(* CODESYS project PLCTEST.project
   Title: PLCTEST
   Author: Peter
   Version: 0.0.0.13

Project tree, tasks and I/O mapping:
  MyController_1 : TM241CEC24T/U, Schneider Electric, order no. TM241CEC24T/U, version 4.0.6.18
    application Application
      libraries: HMISCU PTOPWM, 2.0.1.4 (Schneider Electric); SM3_Basic, 3.5.3.83 (3S - Smart Software Solutions GmbH); CANmotion Lexium Library, 1.3.1.0 (Schneider Electric)
      task MAST (cyclic, interval 2 ms, priority 15, watchdog 100 ms x 1) calls POU_TEST
      program POU_TEST [ST]
      global variables GVL
      program POU [CFC]
    DI : Digital Inputs, Schneider Electric, version 4.0.6.18
        input  iwDI_IW0 : WORD  // IW0
        input  ibDI_IB1 : BYTE  // IB1
    DQ : Digital Outputs, Schneider Electric, version 4.0.6.18
        output Application.POU_TEST.q0 : BOOL  // QW0.Q0
        output Application.POU_TEST.q1 : BOOL  // QW0.Q1
        output Application.POU_TEST.q2 : BOOL  // QW0.Q2
        output Application.POU_TEST.q0 : BOOL  // QW0.Q4
        output Application.POU_TEST.q1 : BOOL  // QW0.Q5
        output Application.POU_TEST.q2 : BOOL  // QW0.Q6
        output Application.POU_TEST.q0 : BOOL  // QW0.Q8
        output Application.POU_TEST.q1 : BOOL  // QW0.Q9
        unmapped channels: QW0, QB1
    Counters : Counters, Schneider Electric, version 4.0.6.18
    Pulse_Generators : Pulse Generators, Schneider Electric, version 4.0.6.18
    Cartridge_1 : Cartridge, Schneider Electric, version 4.0.6.18
    IO_Bus : IO bus - TM3, Schneider Electric, version 4.0.6.18
      Module_1 : TM3SAF5R/G, Schneider Electric, order no. TM3SAF5R/G, version 1.0.1.12
          input  iwModule_1_IW0 : WORD  // IW0
          output qbModule_1_QB0 : BYTE  // QB0
      Module_2 : TM3AQ4/G, Schneider Electric, order no. TM3AQ4/G, version 1.0.0.12
          output qiModule_2_QW0 : INT  // QW0
          output qiModule_2_QW1 : INT  // QW1
          output qiModule_2_QW2 : INT  // QW2
          output qiModule_2_QW3 : INT  // QW3
          input  ibModule_2_IBStatusQW0 : BYTE  // IBStatusQW0
          input  ibModule_2_IBStatusQW1 : BYTE  // IBStatusQW1
          input  ibModule_2_IBStatusQW2 : BYTE  // IBStatusQW2
          input  ibModule_2_IBStatusQW3 : BYTE  // IBStatusQW3
    COM_Bus : COM bus, Schneider Electric, version 4.0.6.18
    Ethernet_1 : Ethernet Network, Schneider Electric, version 4.0.6.18
    Serial_Line_1 : Serial line, Schneider Electric, version 4.0.6.18
      SoMachine_Network_Manager1 : SoMachine-Network Manager, Schneider Electric, version 4.0.0.2
    Serial_Line_2 : Serial line, Schneider Electric, version 4.0.6.18
      Modbus_Manager1 : Modbus Manager, Schneider Electric, version 4.0.0.2
    CAN_1 : CANopen bus, Schneider Electric, version 4.0.6.18
      CANopen_Performance : CANopen Performance, Schneider Electric, order no. 1806, version 3.0.1.24
          settings: Heartbeat in Milliseconds = 100; ConfigVersion = 50659584
        Lexium_32_M : Lexium 32 M, Schneider Electric, order no. 91200, version 3.5.9.0
            settings: General Options.Optional Device = TRUE; NODEIDSAVED = 1; SDO Timeout = 1000000; Explicit Deactivate PDOs = FALSE; EXPERTSETTINGS = False; Nodeguarding.Guard Time = 100 ms; Heartbeat-Producer Time = 200; PDO 16#1400.COBID = 16#0201; PDO 16#1801.COBID = 16#C0000281; Generic COBID = '$NODEID+16#C0000280'; PDO 16#1802.COBID = 16#C0000381; Generic COBID = '$NODEID+16#C0000380'; PDO 16#1803.COBID = 16#C0000481; Generic COBID = '$NODEID+16#C0000480'; Heartbeat-Consuming1.Heartbeat-Time = 300 ms; Controlword.Subindex = 16#00; Target position.Subindex = 16#00; Controlword.Subindex = 16#00; Target velocity.Subindex = 16#00; Statusword.Subindex = 16#00; Position actual value.Subindex = 16#00; Statusword.Subindex = 16#00; Velocity actual value.Subindex = 16#00; SDO List.Set Guardtime.Index = 16#100C; SDO List.Set Guardtime.Subindex = 16#00; SDO List.Set Guardtime.Value = 16#00000064; SDO List.Set Guardtime.Size = 16; SDO List.Set Guardtime.AbortIfError = FALSE; SDO List.Set Guardtime.JumpToLine = FALSE; SDO List.Set Guardtime.Line = 0; SDO List.Set Lifetime.Index = 16#100D; SDO List.Set Lifetime.Subindex = 16#00; SDO List.Set Lifetime.Value = 16#00000000; SDO List.Set Lifetime.Size = 8; SDO List.Set Lifetime.AbortIfError = FALSE; SDO List.Set Lifetime.JumpToLine = FALSE; SDO List.Set Lifetime.Line = 0; SDO List.Disable Emcy CobID.Index = 16#1014; SDO List.Disable Emcy CobID.Subindex = 16#00; SDO List.Disable Emcy CobID.Value = 16#80000081;
              SDO List.Disable Emcy CobID.Size = 32; SDO List.Disable Emcy CobID.AbortIfError = FALSE; SDO List.Disable Emcy CobID.JumpToLine = FALSE; SDO List.Disable Emcy CobID.Line = 0; SDO List.Set Emcy CobID.Index = 16#1014; SDO List.Set Emcy CobID.Subindex = 16#00; SDO List.Set Emcy CobID.Value = 16#00000081; SDO List.Set Emcy CobID.Size = 32; SDO List.Set Emcy CobID.AbortIfError = FALSE; SDO List.Set Emcy CobID.JumpToLine = FALSE; SDO List.Set Emcy CobID.Line = 0; SDO List.Set Heartbeat Consumer.Index = 16#1016; SDO List.Set Heartbeat Consumer.Subindex = 16#01; SDO List.Set Heartbeat Consumer.Value = 16#007F012C; SDO List.Set Heartbeat Consumer.Size = 32; SDO List.Set Heartbeat Consumer.AbortIfError = FALSE; SDO List.Set Heartbeat Consumer.JumpToLine = FALSE; SDO List.Set Heartbeat Consumer.Line = 0; SDO List.Set Heartbeat Consumer.Index = 16#1016; SDO List.Set Heartbeat Consumer.Subindex = 16#02; SDO List.Set Heartbeat Consumer.Value = 0; SDO List.Set Heartbeat Consumer.Size = 32; SDO List.Set Heartbeat Consumer.AbortIfError = FALSE; SDO List.Set Heartbeat Consumer.JumpToLine = FALSE; SDO List.Set Heartbeat Consumer.Line = 0; SDO List.Set Heartbeat Consumer.Index = 16#1016; SDO List.Set Heartbeat Consumer.Subindex = 16#03; SDO List.Set Heartbeat Consumer.Value = 0; SDO List.Set Heartbeat Consumer.Size = 32; SDO List.Set Heartbeat Consumer.AbortIfError = FALSE; SDO List.Set Heartbeat Consumer.JumpToLine = FALSE; SDO List.Set Heartbeat Consumer.Line = 0; SDO List.Set Heartbeat Producer.Index = 16#1017; SDO List.Set Heartbeat Producer.Subindex = 16#00; SDO List.Set Heartbeat Producer.Value = 16#000000C8; SDO List.Set Heartbeat Producer.Size = 16; SDO List.Set Heartbeat Producer.AbortIfError = FALSE; SDO List.Set Heartbeat Producer.JumpToLine = FALSE; SDO List.Set Heartbeat Producer.Line = 0; SDO List.Disable PDO.Index = 16#1400;
              SDO List.Disable PDO.Subindex = 16#01; SDO List.Disable PDO.Value = 16#80000201; SDO List.Disable PDO.Size = 32; SDO List.Disable PDO.AbortIfError = FALSE; SDO List.Disable PDO.JumpToLine = FALSE; SDO List.Disable PDO.Line = 0; SDO List.Set transmission type.Index = 16#1400; SDO List.Set transmission type.Subindex = 16#02; SDO List.Set transmission type.Value = 16#FF; SDO List.Set transmission type.Size = 8; SDO List.Set transmission type.AbortIfError = FALSE; SDO List.Set transmission type.JumpToLine = FALSE; SDO List.Set transmission type.Line = 0; SDO List.Clear pdo mapping.Index = 16#1600; SDO List.Clear pdo mapping.Subindex = 16#00; SDO List.Clear pdo mapping.Value = 16#0; SDO List.Clear pdo mapping.Size = 8; SDO List.Clear pdo mapping.AbortIfError = FALSE; SDO List.Clear pdo mapping.JumpToLine = FALSE; SDO List.Clear pdo mapping.Line = 0; SDO List.Set Mapping.Index = 16#1600; SDO List.Set Mapping.Subindex = 16#01; SDO List.Set Mapping.Value = 16#301B1F10; SDO List.Set Mapping.Size = 32; SDO List.Set Mapping.AbortIfError = FALSE; SDO List.Set Mapping.JumpToLine = FALSE; SDO List.Set Mapping.Line = 0; SDO List.Set Mapping.Index = 16#1600; SDO List.Set Mapping.Subindex = 16#02; SDO List.Set Mapping.Value = 16#301B2210; SDO List.Set Mapping.Size = 32; SDO List.Set Mapping.AbortIfError = FALSE; SDO List.Set Mapping.JumpToLine = FALSE; SDO List.Set Mapping.Line = 0; SDO List.Set Mapping.Index = 16#1600; SDO List.Set Mapping.Subindex = 16#03; SDO List.Set Mapping.Value = 16#301B2120; SDO List.Set Mapping.Size = 32; SDO List.Set Mapping.AbortIfError = FALSE; SDO List.Set Mapping.JumpToLine = FALSE;
              SDO List.Set Mapping.Line = 0; SDO List.Set number of pdos.Index = 16#1600; SDO List.Set number of pdos.Subindex = 16#00; SDO List.Set number of pdos.Value = 16#03; SDO List.Set number of pdos.Size = 8; SDO List.Set number of pdos.AbortIfError = FALSE; SDO List.Set number of pdos.JumpToLine = FALSE; SDO List.Set number of pdos.Line = 0; SDO List.Set and enable COB-ID.Index = 16#1400; SDO List.Set and enable COB-ID.Subindex = 16#01; SDO List.Set and enable COB-ID.Value = 16#00000201; SDO List.Set and enable COB-ID.Size = 32; SDO List.Set and enable COB-ID.AbortIfError = FALSE; SDO List.Set and enable COB-ID.JumpToLine = FALSE; SDO List.Set and enable COB-ID.Line = 0; SDO List.Disable PDO.Index = 16#1401; SDO List.Disable PDO.Subindex = 16#01; SDO List.Disable PDO.Value = 16#80000301; SDO List.Disable PDO.Size = 32; SDO List.Disable PDO.AbortIfError = FALSE; SDO List.Disable PDO.JumpToLine = FALSE; SDO List.Disable PDO.Line = 0; SDO List.Disable PDO.Index = 16#1402; SDO List.Disable PDO.Subindex = 16#01; SDO List.Disable PDO.Value = 16#80000401; SDO List.Disable PDO.Size = 32; SDO List.Disable PDO.AbortIfError = FALSE; SDO List.Disable PDO.JumpToLine = FALSE; SDO List.Disable PDO.Line = 0; SDO List.Disable PDO.Index = 16#1403; SDO List.Disable PDO.Subindex = 16#01; SDO List.Disable PDO.Value = 16#80000501; SDO List.Disable PDO.Size = 32; SDO List.Disable PDO.AbortIfError = FALSE; SDO List.Disable PDO.JumpToLine = FALSE; SDO List.Disable PDO.Line = 0; SDO List.Disable PDO.Index = 16#1800; SDO List.Disable PDO.Subindex = 16#01; SDO List.Disable PDO.Value = 16#C0000181; SDO List.Disable PDO.Size = 32;
              SDO List.Disable PDO.AbortIfError = FALSE; SDO List.Disable PDO.JumpToLine = FALSE; SDO List.Disable PDO.Line = 0; SDO List.Set transmission type.Index = 16#1800; SDO List.Set transmission type.Subindex = 16#02; SDO List.Set transmission type.Value = 16#FF; SDO List.Set transmission type.Size = 8; SDO List.Set transmission type.AbortIfError = FALSE; SDO List.Set transmission type.JumpToLine = FALSE; SDO List.Set transmission type.Line = 0; SDO List.Set inhibit time.Index = 16#1800; SDO List.Set inhibit time.Subindex = 16#03; SDO List.Set inhibit time.Value = 16#0064; SDO List.Set inhibit time.Size = 16; SDO List.Set inhibit time.AbortIfError = FALSE; SDO List.Set inhibit time.JumpToLine = FALSE; SDO List.Set inhibit time.Line = 0; SDO List.Set event time.Index = 16#1800; SDO List.Set event time.Subindex = 16#05; SDO List.Set event time.Value = 16#0000; SDO List.Set event time.Size = 16; SDO List.Set event time.AbortIfError = FALSE; SDO List.Set event time.JumpToLine = FALSE; SDO List.Set event time.Line = 0; SDO List.Clear pdo mapping.Index = 16#1A00; SDO List.Clear pdo mapping.Subindex = 16#00; SDO List.Clear pdo mapping.Value = 16#0; SDO List.Clear pdo mapping.Size = 8; SDO List.Clear pdo mapping.AbortIfError = FALSE; SDO List.Clear pdo mapping.JumpToLine = FALSE; SDO List.Clear pdo mapping.Line = 0; SDO List.Set Mapping.Index = 16#1A00; SDO List.Set Mapping.Subindex = 16#01; SDO List.Set Mapping.Value = 16#301B2510; SDO List.Set Mapping.Size = 32; SDO List.Set Mapping.AbortIfError = FALSE; SDO List.Set Mapping.JumpToLine = FALSE; SDO List.Set Mapping.Line = 0; SDO List.Set Mapping.Index = 16#1A00; SDO List.Set Mapping.Subindex = 16#02;
              SDO List.Set Mapping.Value = 16#301B2610; SDO List.Set Mapping.Size = 32; SDO List.Set Mapping.AbortIfError = FALSE; SDO List.Set Mapping.JumpToLine = FALSE; SDO List.Set Mapping.Line = 0; SDO List.Set Mapping.Index = 16#1A00; SDO List.Set Mapping.Subindex = 16#03; SDO List.Set Mapping.Value = 16#301B2710; SDO List.Set Mapping.Size = 32; SDO List.Set Mapping.AbortIfError = FALSE; SDO List.Set Mapping.JumpToLine = FALSE; SDO List.Set Mapping.Line = 0; SDO List.Set Mapping.Index = 16#1A00; SDO List.Set Mapping.Subindex = 16#04; SDO List.Set Mapping.Value = 16#301B2810; SDO List.Set Mapping.Size = 32; SDO List.Set Mapping.AbortIfError = FALSE; SDO List.Set Mapping.JumpToLine = FALSE; SDO List.Set Mapping.Line = 0; SDO List.Set number of pdos.Index = 16#1A00; SDO List.Set number of pdos.Subindex = 16#00; SDO List.Set number of pdos.Value = 16#04; SDO List.Set number of pdos.Size = 8; SDO List.Set number of pdos.AbortIfError = FALSE; SDO List.Set number of pdos.JumpToLine = FALSE; SDO List.Set number of pdos.Line = 0; SDO List.Set and enable COB-ID.Index = 16#1800; SDO List.Set and enable COB-ID.Subindex = 16#01; SDO List.Set and enable COB-ID.Value = 16#40000181; SDO List.Set and enable COB-ID.Size = 32; SDO List.Set and enable COB-ID.AbortIfError = FALSE; SDO List.Set and enable COB-ID.JumpToLine = FALSE; SDO List.Set and enable COB-ID.Line = 0; SDO List.Disable PDO.Index = 16#1801; SDO List.Disable PDO.Subindex = 16#01; SDO List.Disable PDO.Value = 16#C0000281; SDO List.Disable PDO.Size = 32; SDO List.Disable PDO.AbortIfError = FALSE; SDO List.Disable PDO.JumpToLine = FALSE; SDO List.Disable PDO.Line = 0;
              SDO List.Disable PDO.Index = 16#1802; SDO List.Disable PDO.Subindex = 16#01; SDO List.Disable PDO.Value = 16#C0000381; SDO List.Disable PDO.Size = 32; SDO List.Disable PDO.AbortIfError = FALSE; SDO List.Disable PDO.JumpToLine = FALSE; SDO List.Disable PDO.Line = 0; SDO List.Disable PDO.Index = 16#1803; SDO List.Disable PDO.Subindex = 16#01; SDO List.Disable PDO.Value = 16#C0000481; SDO List.Disable PDO.Size = 32; SDO List.Disable PDO.AbortIfError = FALSE; SDO List.Disable PDO.JumpToLine = FALSE; SDO List.Disable PDO.Line = 0; SDO List.Automap SDO1.Index = 16#3041; SDO List.Automap SDO1.Subindex = 16#0B; SDO List.Automap SDO1.Value = 15; SDO List.Automap SDO1.Size = 16; SDO List.Automap SDO1.AbortIfError = FALSE; SDO List.Automap SDO1.JumpToLine = FALSE; SDO List.Automap SDO1.Line = 0; SDO List.Automap SDO2.Index = 16#301B; SDO List.Automap SDO2.Subindex = 16#08; SDO List.Automap SDO2.Value = 1; SDO List.Automap SDO2.Size = 16; SDO List.Automap SDO2.AbortIfError = FALSE; SDO List.Automap SDO2.JumpToLine = FALSE; SDO List.Automap SDO2.Line = 0; SDO List.Automap SDO2.Index = 16#301B; SDO List.Automap SDO2.Subindex = 16#1E; SDO List.Automap SDO2.Value = 10; SDO List.Automap SDO2.Size = 16; SDO List.Automap SDO2.AbortIfError = FALSE; SDO List.Automap SDO2.JumpToLine = FALSE; SDO List.Automap SDO2.Line = 0; ConfigVersion = 50659584
            unmapped channels: driveModeCtrl, RefA16, RefB32, driveStat, mfStat, motionStat, driveInput
*)

// MyController_1/Application/GVL
VAR_GLOBAL
END_VAR

// MyController_1/Application/POU_TEST
PROGRAM POU_TEST
VAR
	power_: INT;
	counter : INT := 0;
	lights : ARRAY [0..3] OF BOOL;
	q0 : BOOL;
	q1 : BOOL;
	q2 : BOOL;
	execute : BOOL;
	
	limit_1 : SEM_LXM.SetLimitSwitch_LXM;
	limit_2 : SEM_LXM.SetLimitSwitch_LXM;
	
	
	wordName : WORD;

	powerLXM : MC_Power_LXM;
	//power : SM3_Basic.MC_Power;
	motorJog : MC_Jog_LXM;
	mcReadParameter : MC_ReadAxisError_LXM;
	resetLXM : SEM_LXM.MC_Reset_LXM;
	power_1 : SEM_LXM.MC_Power_LXM;
	//stop : SM3_Basic.MC_Stop;
	//home : SM3_Basic.MC_Home;
	
	
	
	
	testOut :BOOL;


END_VAR

(*
//power.Enable := TRUE;
(*
powerLXM.Axis := Lexium_32_M;
motorJog.Axis := Lexium_32_M;*)
q0 := TRUE;
//resetLXM.

powerLXM.Enable := TRUE;
motorJog.Forward := TRUE;


//home.Execute:= TRUE;
powerLXM(Axis := Lexium_32_M);
//stop();
motorJog(Axis := Lexium_32_M);

*)
qbModule_1_QB0 := 0001;

mcReadParameter.Enable := TRUE;

wordName := mcReadParameter.ErrorID;
power_1.Enable := TRUE;

q1 := TRUE;

mcReadParameter(Axis := Lexium_32_M);

power_1(Axis := Lexium_32_M);
limit_1.LimitSwitch := 1;
limit_1.Mode := 0;

limit_1.Execute := execute;
limit_1(Axis := Lexium_32_M);

limit_2.LimitSwitch := 2;
limit_2.Mode := 0;
limit_2.Execute := execute;
limit_2(Axis := Lexium_32_M);

resetLXM(Axis := Lexium_32_M);



//motorJog.Forward := TRUE;
//motorJog.Fast := TRUE;
//motorJog.TipPos := 100;

motorJog(Axis := Lexium_32_M);

END_PROGRAM

// MyController_1/Application/POU
PROGRAM POU
VAR
	MC_Power_LXM_0: MC_Power_LXM;
	MC_ReadActualVelocity_LXM_0: MC_ReadActualVelocity_LXM;
	MC_MoveVelocity_LXM_0: MC_MoveVelocity_LXM;
	MC_Reset_LXM_0: MC_Reset_LXM;
	MC_ReadStatus_LXM_0 : MC_ReadStatus_LXM;
	xPower: BOOL;
	xReset: BOOL;
	MC_Stop_LXM_0: MC_Stop_LXM;
	xStop: BOOL;
	xMove: BOOL;
END_VAR

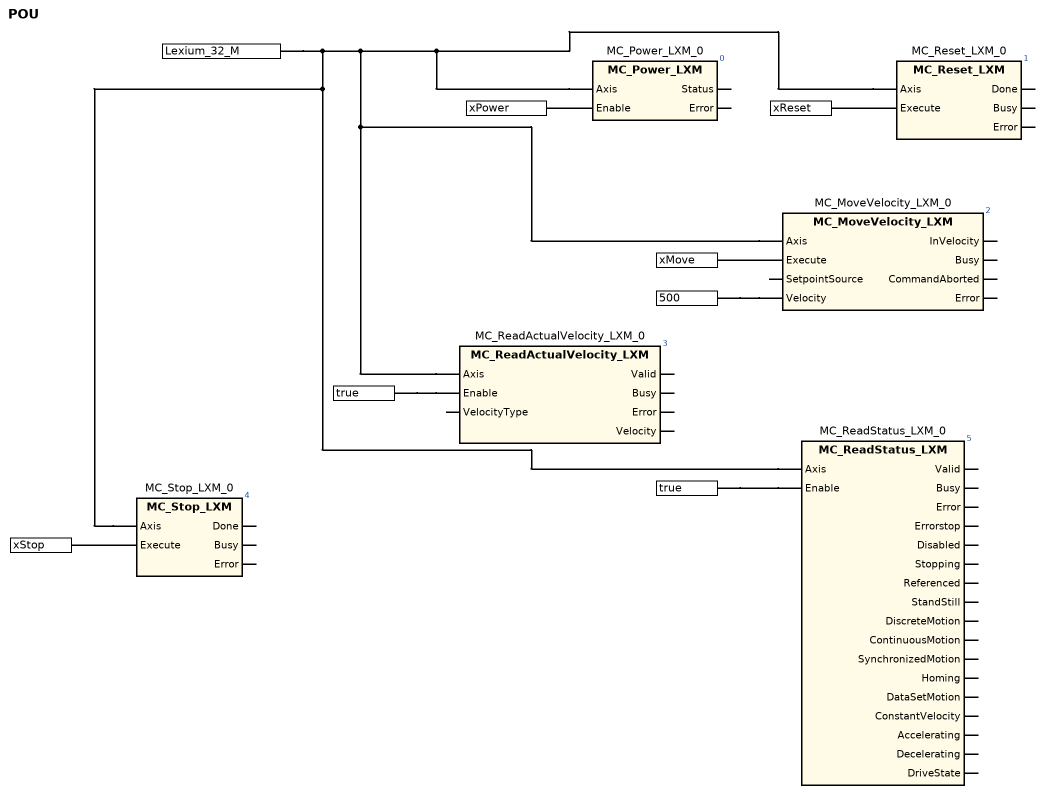
MC_Power_LXM_0(Axis := Lexium_32_M, Enable := xPower); // MC_Power_LXM
MC_Reset_LXM_0(Axis := Lexium_32_M, Execute := xReset); // MC_Reset_LXM
MC_MoveVelocity_LXM_0(Axis := Lexium_32_M, Execute := xMove, Velocity := 500); // MC_MoveVelocity_LXM
MC_ReadActualVelocity_LXM_0(Axis := Lexium_32_M, Enable := true); // MC_ReadActualVelocity_LXM
MC_Stop_LXM_0(Axis := Lexium_32_M, Execute := xStop); // MC_Stop_LXM
MC_ReadStatus_LXM_0(Axis := Lexium_32_M, Enable := true); // MC_ReadStatus_LXM

END_PROGRAM
